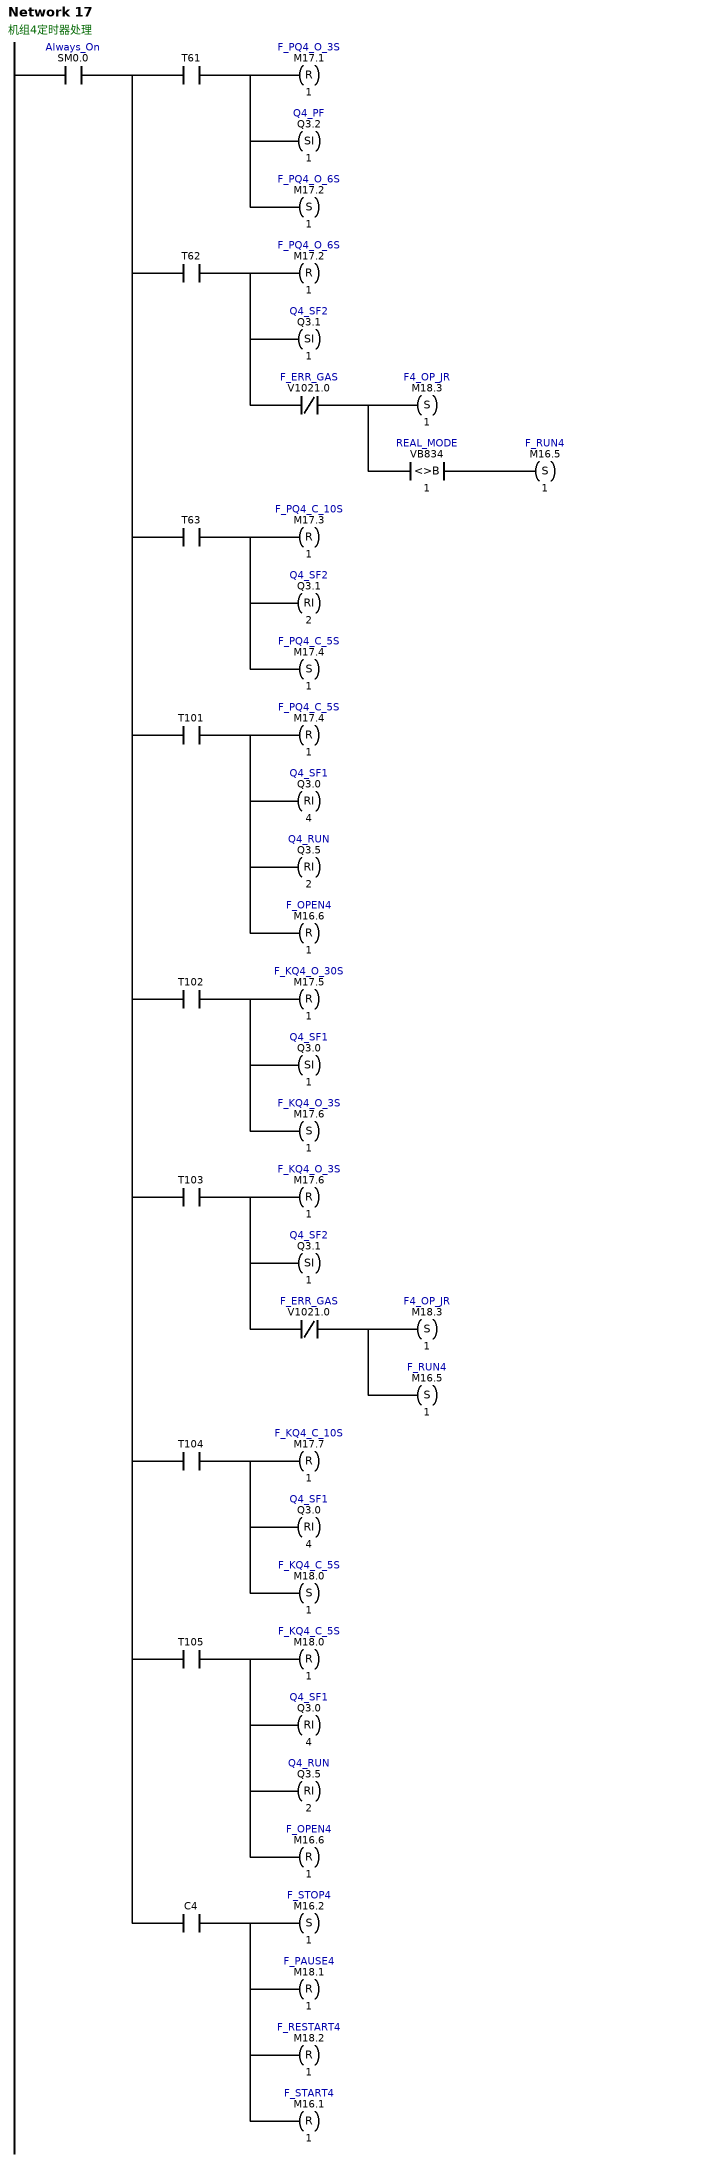
[picture p72: SBR7 networks 17-17]
Network 17
// 机组4定时器处理
LD     Always_On:SM0.0
LPS
A      T61
R      F_PQ4_O_3S:M17.1, 1
SI     Q4_PF:Q3.2, 1
S      F_PQ4_O_6S:M17.2, 1
LRD
A      T62
R      F_PQ4_O_6S:M17.2, 1
SI     Q4_SF2:Q3.1, 1
AN     F_ERR_GAS:V1021.0
S      F4_OP_JR:M18.3, 1
AB<>   REAL_MODE:VB834, 1
S      F_RUN4:M16.5, 1
LRD
LPS
A      T63
R      F_PQ4_C_10S:M17.3, 1
RI     Q4_SF2:Q3.1, 2
S      F_PQ4_C_5S:M17.4, 1
LRD
A      T101
R      F_PQ4_C_5S:M17.4, 1
RI     Q4_SF1:Q3.0, 4
RI     Q4_RUN:Q3.5, 2
R      F_OPEN4:M16.6, 1
LPP
A      T102
R      F_KQ4_O_30S:M17.5, 1
SI     Q4_SF1:Q3.0, 1
S      F_KQ4_O_3S:M17.6, 1
LRD
A      T103
R      F_KQ4_O_3S:M17.6, 1
SI     Q4_SF2:Q3.1, 1
AN     F_ERR_GAS:V1021.0
S      F4_OP_JR:M18.3, 1
S      F_RUN4:M16.5, 1
LPP
LPS
A      T104
R      F_KQ4_C_10S:M17.7, 1
RI     Q4_SF1:Q3.0, 4
S      F_KQ4_C_5S:M18.0, 1
LRD
A      T105
R      F_KQ4_C_5S:M18.0, 1
RI     Q4_SF1:Q3.0, 4
RI     Q4_RUN:Q3.5, 2
R      F_OPEN4:M16.6, 1
LPP
A      C4
S      F_STOP4:M16.2, 1
R      F_PAUSE4:M18.1, 1
R      F_RESTART4:M18.2, 1
R      F_START4:M16.1, 1
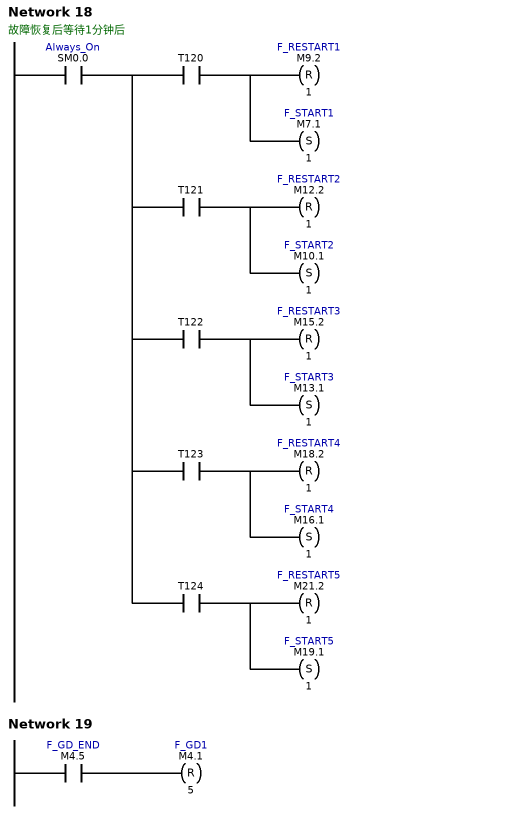
Network 18
// 故障恢复后等待1分钟后
LD     Always_On:SM0.0
LPS
A      T120
R      F_RESTART1:M9.2, 1
S      F_START1:M7.1, 1
LRD
A      T121
R      F_RESTART2:M12.2, 1
S      F_START2:M10.1, 1
LRD
A      T122
R      F_RESTART3:M15.2, 1
S      F_START3:M13.1, 1
LRD
A      T123
R      F_RESTART4:M18.2, 1
S      F_START4:M16.1, 1
LPP
A      T124
R      F_RESTART5:M21.2, 1
S      F_START5:M19.1, 1
Network 19
LD     F_GD_END:M4.5
R      F_GD1:M4.1, 5
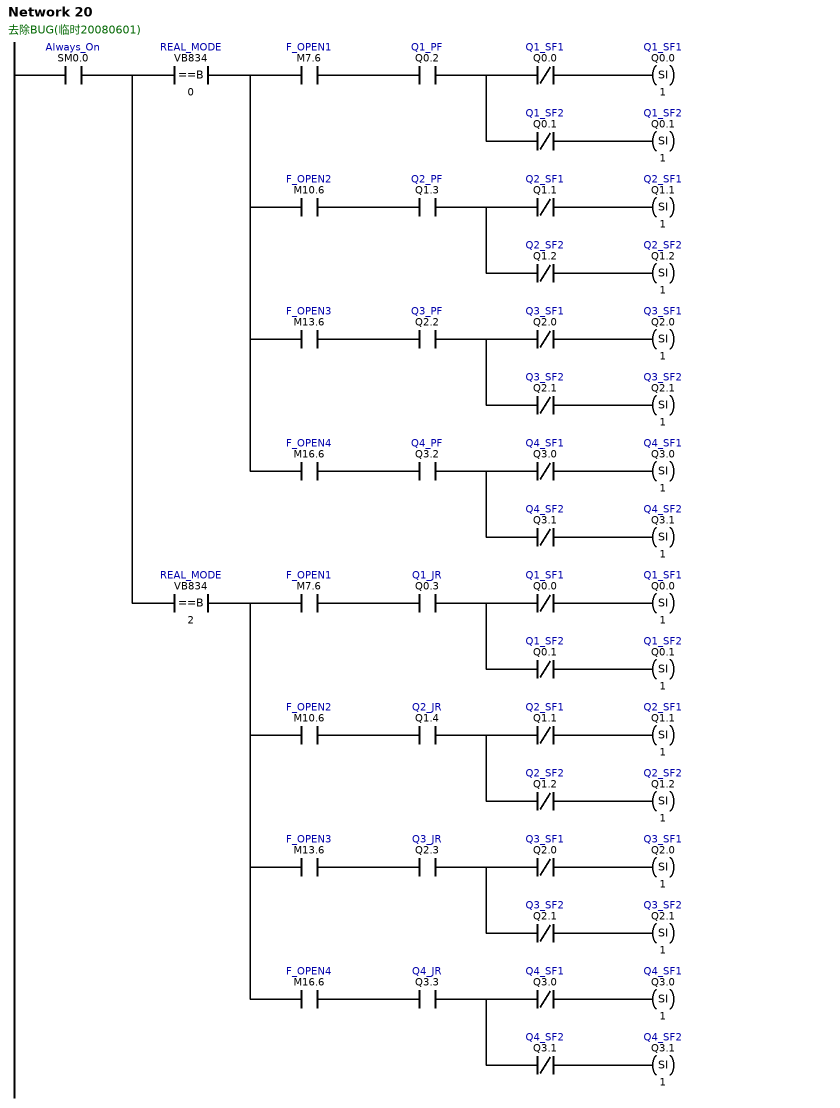
Network 20
// 去除BUG(临时20080601)
LD     Always_On:SM0.0
LPS
AB=    REAL_MODE:VB834, 0
LPS
A      F_OPEN1:M7.6
A      Q1_PF:Q0.2
LPS
AN     Q1_SF1:Q0.0
SI     Q1_SF1:Q0.0, 1
LPP
AN     Q1_SF2:Q0.1
SI     Q1_SF2:Q0.1, 1
LRD
A      F_OPEN2:M10.6
A      Q2_PF:Q1.3
LPS
AN     Q2_SF1:Q1.1
SI     Q2_SF1:Q1.1, 1
LPP
AN     Q2_SF2:Q1.2
SI     Q2_SF2:Q1.2, 1
LRD
A      F_OPEN3:M13.6
A      Q3_PF:Q2.2
LPS
AN     Q3_SF1:Q2.0
SI     Q3_SF1:Q2.0, 1
LPP
AN     Q3_SF2:Q2.1
SI     Q3_SF2:Q2.1, 1
LPP
A      F_OPEN4:M16.6
A      Q4_PF:Q3.2
LPS
AN     Q4_SF1:Q3.0
SI     Q4_SF1:Q3.0, 1
LPP
AN     Q4_SF2:Q3.1
SI     Q4_SF2:Q3.1, 1
LPP
AB=    REAL_MODE:VB834, 2
LPS
A      F_OPEN1:M7.6
A      Q1_JR:Q0.3
LPS
AN     Q1_SF1:Q0.0
SI     Q1_SF1:Q0.0, 1
LPP
AN     Q1_SF2:Q0.1
SI     Q1_SF2:Q0.1, 1
LRD
A      F_OPEN2:M10.6
A      Q2_JR:Q1.4
LPS
AN     Q2_SF1:Q1.1
SI     Q2_SF1:Q1.1, 1
LPP
AN     Q2_SF2:Q1.2
SI     Q2_SF2:Q1.2, 1
LRD
A      F_OPEN3:M13.6
A      Q3_JR:Q2.3
LPS
AN     Q3_SF1:Q2.0
SI     Q3_SF1:Q2.0, 1
LPP
AN     Q3_SF2:Q2.1
SI     Q3_SF2:Q2.1, 1
LPP
A      F_OPEN4:M16.6
A      Q4_JR:Q3.3
LPS
AN     Q4_SF1:Q3.0
SI     Q4_SF1:Q3.0, 1
LPP
AN     Q4_SF2:Q3.1
SI     Q4_SF2:Q3.1, 1
END_SUBROUTINE_BLOCK

SUBROUTINE_BLOCK 读EEPROM:SBR8
TITLE=
VAR
TEMP:DWORD;	// LD0 
END_VAR
BEGIN
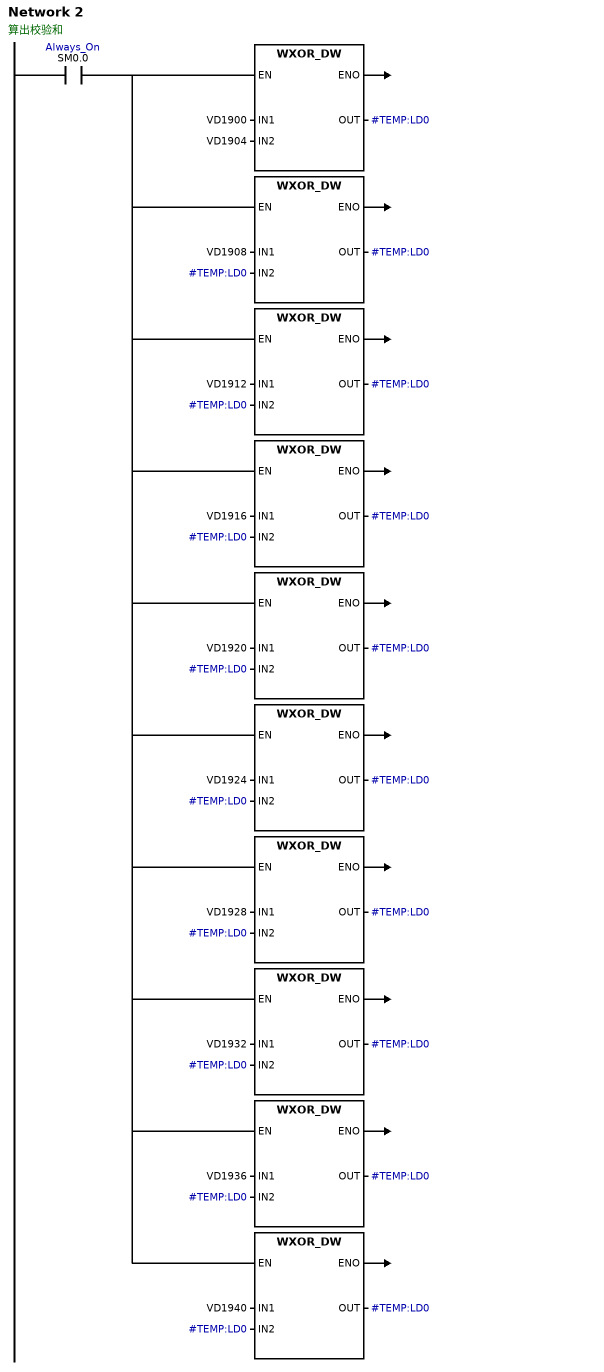
Network 2
// 算出校验和
LD     Always_On:SM0.0
MOVD   VD1900, #TEMP:LD0
XORD   VD1904, #TEMP:LD0
XORD   VD1908, #TEMP:LD0
XORD   VD1912, #TEMP:LD0
XORD   VD1916, #TEMP:LD0
XORD   VD1920, #TEMP:LD0
XORD   VD1924, #TEMP:LD0
XORD   VD1928, #TEMP:LD0
XORD   VD1932, #TEMP:LD0
XORD   VD1936, #TEMP:LD0
XORD   VD1940, #TEMP:LD0
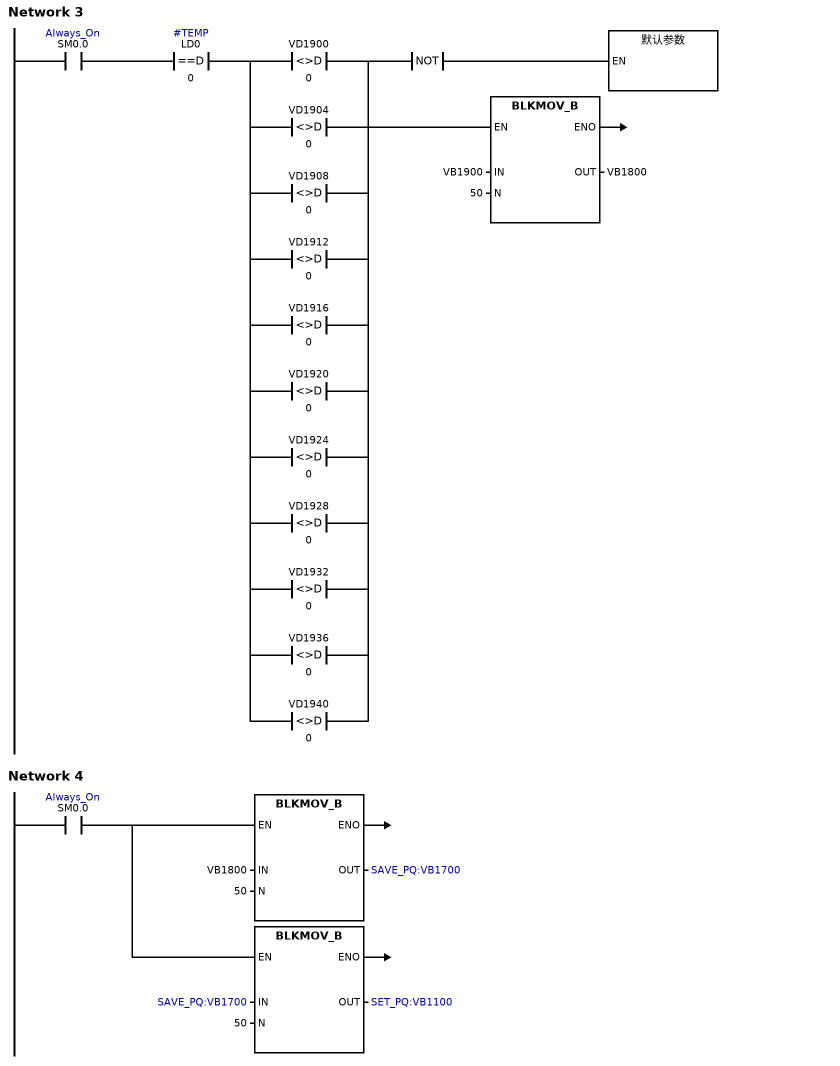
Network 3
LD     Always_On:SM0.0
AD=    #TEMP:LD0, 0
LDD<>  VD1900, 0
OD<>   VD1904, 0
OD<>   VD1908, 0
OD<>   VD1912, 0
OD<>   VD1916, 0
OD<>   VD1920, 0
OD<>   VD1924, 0
OD<>   VD1928, 0
OD<>   VD1932, 0
OD<>   VD1936, 0
OD<>   VD1940, 0
ALD
LPS
NOT
CALL   默认参数:SBR21
LPP
BMB    VB1900, VB1800, 50
Network 4
LD     Always_On:SM0.0
BMB    VB1800, SAVE_PQ:VB1700, 50
BMB    SAVE_PQ:VB1700, SET_PQ:VB1100, 50
END_SUBROUTINE_BLOCK

SUBROUTINE_BLOCK 定时器:SBR9
TITLE=
VAR
TEMP_W:WORD;	// LW0 
END_VAR
BEGIN
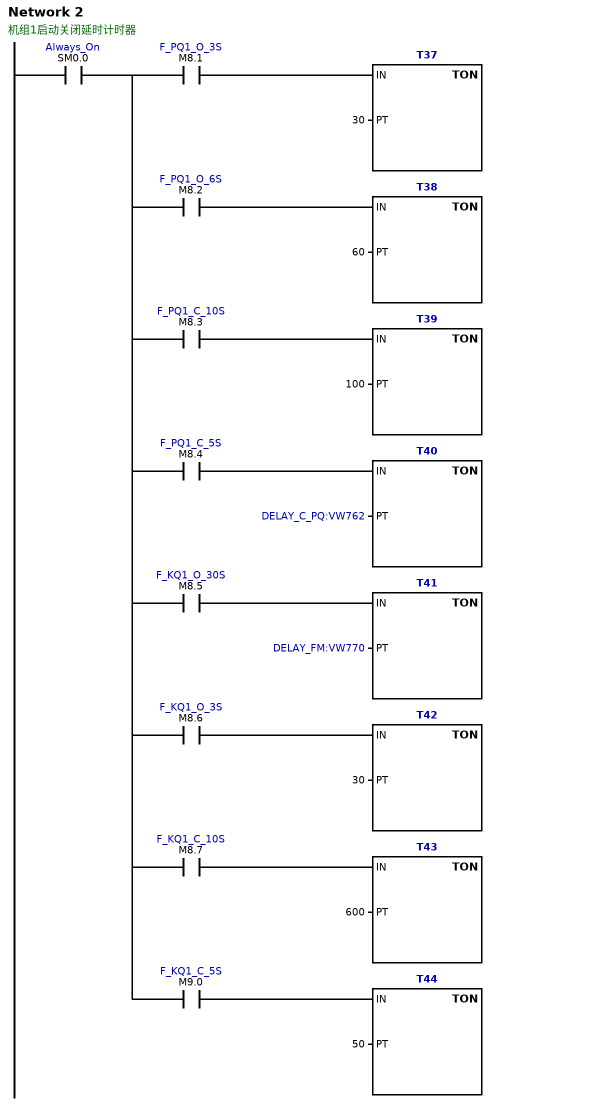
Network 2
// 机组1启动关闭延时计时器
LD     Always_On:SM0.0
LPS
A      F_PQ1_O_3S:M8.1
TON    T37, 30
LRD
A      F_PQ1_O_6S:M8.2
TON    T38, 60
LRD
A      F_PQ1_C_10S:M8.3
TON    T39, 100
LRD
A      F_PQ1_C_5S:M8.4
TON    T40, DELAY_C_PQ:VW762
LRD
A      F_KQ1_O_30S:M8.5
TON    T41, DELAY_FM:VW770
LRD
A      F_KQ1_O_3S:M8.6
TON    T42, 30
LRD
A      F_KQ1_C_10S:M8.7
TON    T43, 600
LPP
A      F_KQ1_C_5S:M9.0
TON    T44, 50
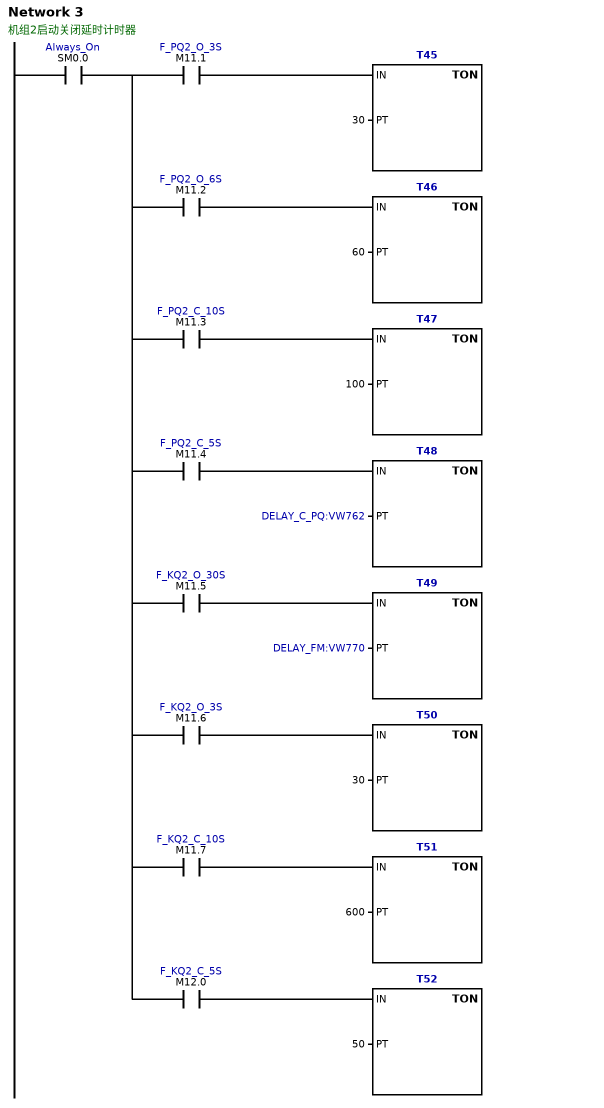
Network 3
// 机组2启动关闭延时计时器
LD     Always_On:SM0.0
LPS
A      F_PQ2_O_3S:M11.1
TON    T45, 30
LRD
A      F_PQ2_O_6S:M11.2
TON    T46, 60
LRD
A      F_PQ2_C_10S:M11.3
TON    T47, 100
LRD
A      F_PQ2_C_5S:M11.4
TON    T48, DELAY_C_PQ:VW762
LRD
A      F_KQ2_O_30S:M11.5
TON    T49, DELAY_FM:VW770
LRD
A      F_KQ2_O_3S:M11.6
TON    T50, 30
LRD
A      F_KQ2_C_10S:M11.7
TON    T51, 600
LPP
A      F_KQ2_C_5S:M12.0
TON    T52, 50
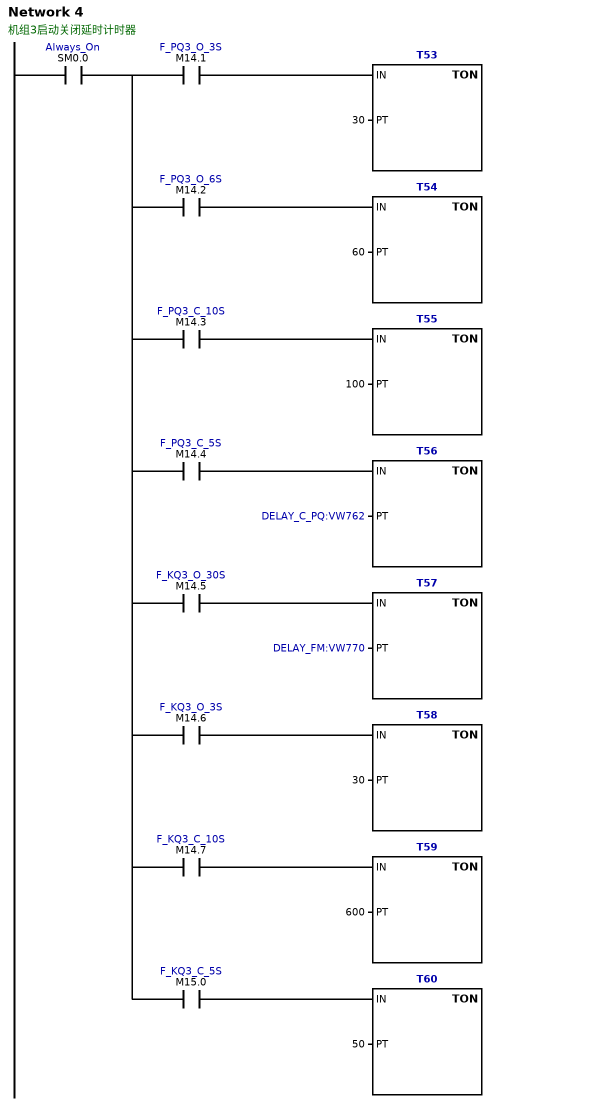
Network 4
// 机组3启动关闭延时计时器
LD     Always_On:SM0.0
LPS
A      F_PQ3_O_3S:M14.1
TON    T53, 30
LRD
A      F_PQ3_O_6S:M14.2
TON    T54, 60
LRD
A      F_PQ3_C_10S:M14.3
TON    T55, 100
LRD
A      F_PQ3_C_5S:M14.4
TON    T56, DELAY_C_PQ:VW762
LRD
A      F_KQ3_O_30S:M14.5
TON    T57, DELAY_FM:VW770
LRD
A      F_KQ3_O_3S:M14.6
TON    T58, 30
LRD
A      F_KQ3_C_10S:M14.7
TON    T59, 600
LPP
A      F_KQ3_C_5S:M15.0
TON    T60, 50
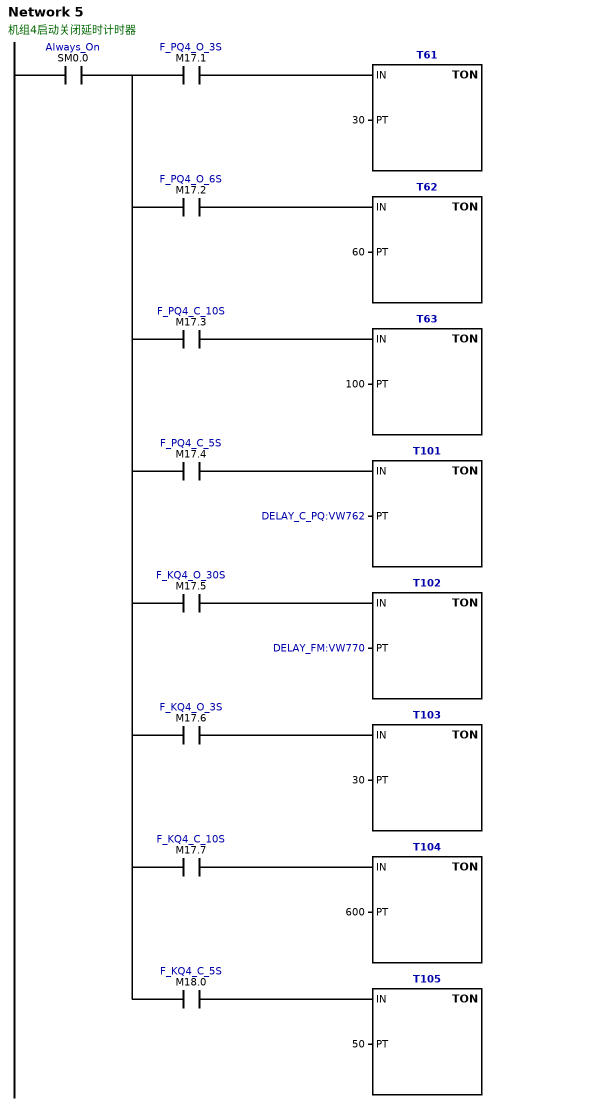
Network 5
// 机组4启动关闭延时计时器
LD     Always_On:SM0.0
LPS
A      F_PQ4_O_3S:M17.1
TON    T61, 30
LRD
A      F_PQ4_O_6S:M17.2
TON    T62, 60
LRD
A      F_PQ4_C_10S:M17.3
TON    T63, 100
LRD
A      F_PQ4_C_5S:M17.4
TON    T101, DELAY_C_PQ:VW762
LRD
A      F_KQ4_O_30S:M17.5
TON    T102, DELAY_FM:VW770
LRD
A      F_KQ4_O_3S:M17.6
TON    T103, 30
LRD
A      F_KQ4_C_10S:M17.7
TON    T104, 600
LPP
A      F_KQ4_C_5S:M18.0
TON    T105, 50
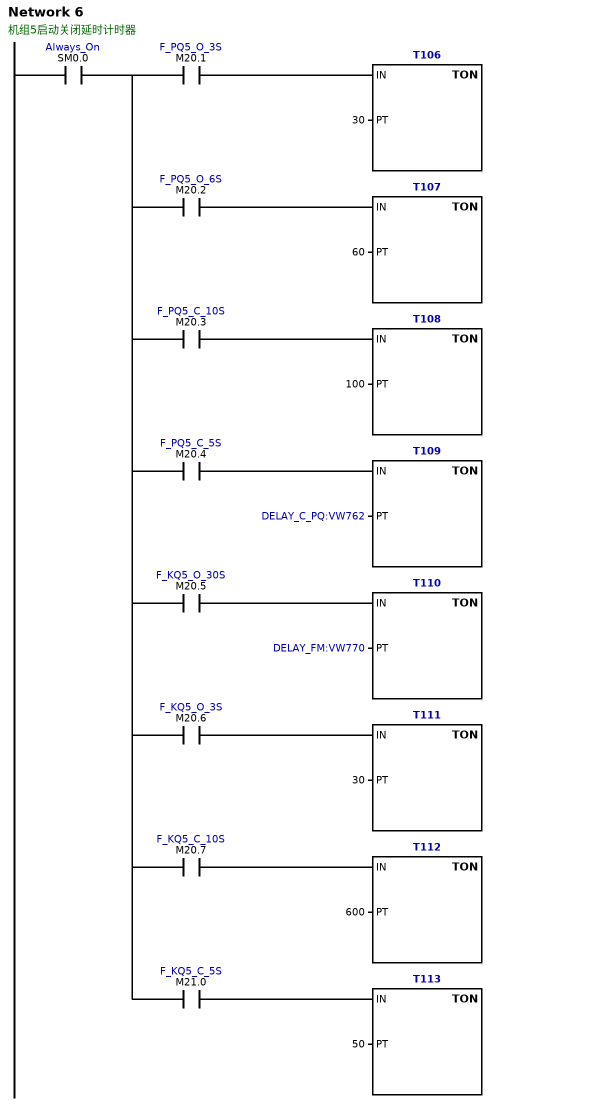
Network 6
// 机组5启动关闭延时计时器
LD     Always_On:SM0.0
LPS
A      F_PQ5_O_3S:M20.1
TON    T106, 30
LRD
A      F_PQ5_O_6S:M20.2
TON    T107, 60
LRD
A      F_PQ5_C_10S:M20.3
TON    T108, 100
LRD
A      F_PQ5_C_5S:M20.4
TON    T109, DELAY_C_PQ:VW762
LRD
A      F_KQ5_O_30S:M20.5
TON    T110, DELAY_FM:VW770
LRD
A      F_KQ5_O_3S:M20.6
TON    T111, 30
LRD
A      F_KQ5_C_10S:M20.7
TON    T112, 600
LPP
A      F_KQ5_C_5S:M21.0
TON    T113, 50
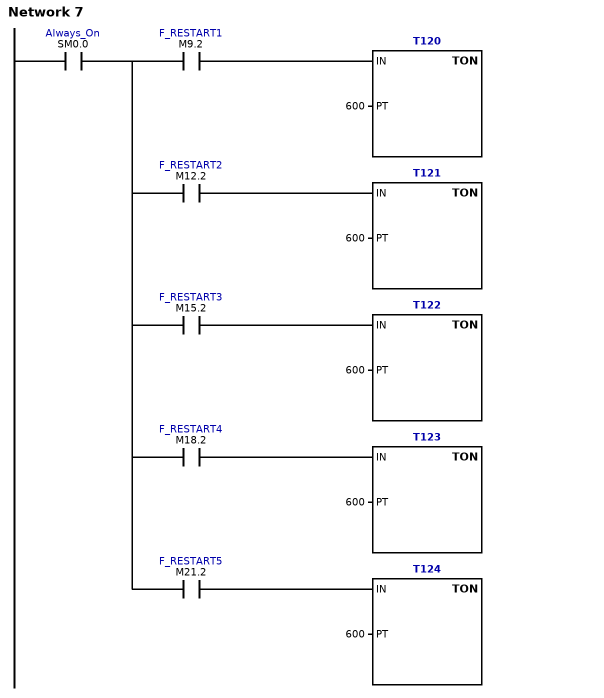
Network 7
LD     Always_On:SM0.0
LPS
A      F_RESTART1:M9.2
TON    T120, 600
LRD
A      F_RESTART2:M12.2
TON    T121, 600
LRD
A      F_RESTART3:M15.2
TON    T122, 600
LRD
A      F_RESTART4:M18.2
TON    T123, 600
LPP
A      F_RESTART5:M21.2
TON    T124, 600
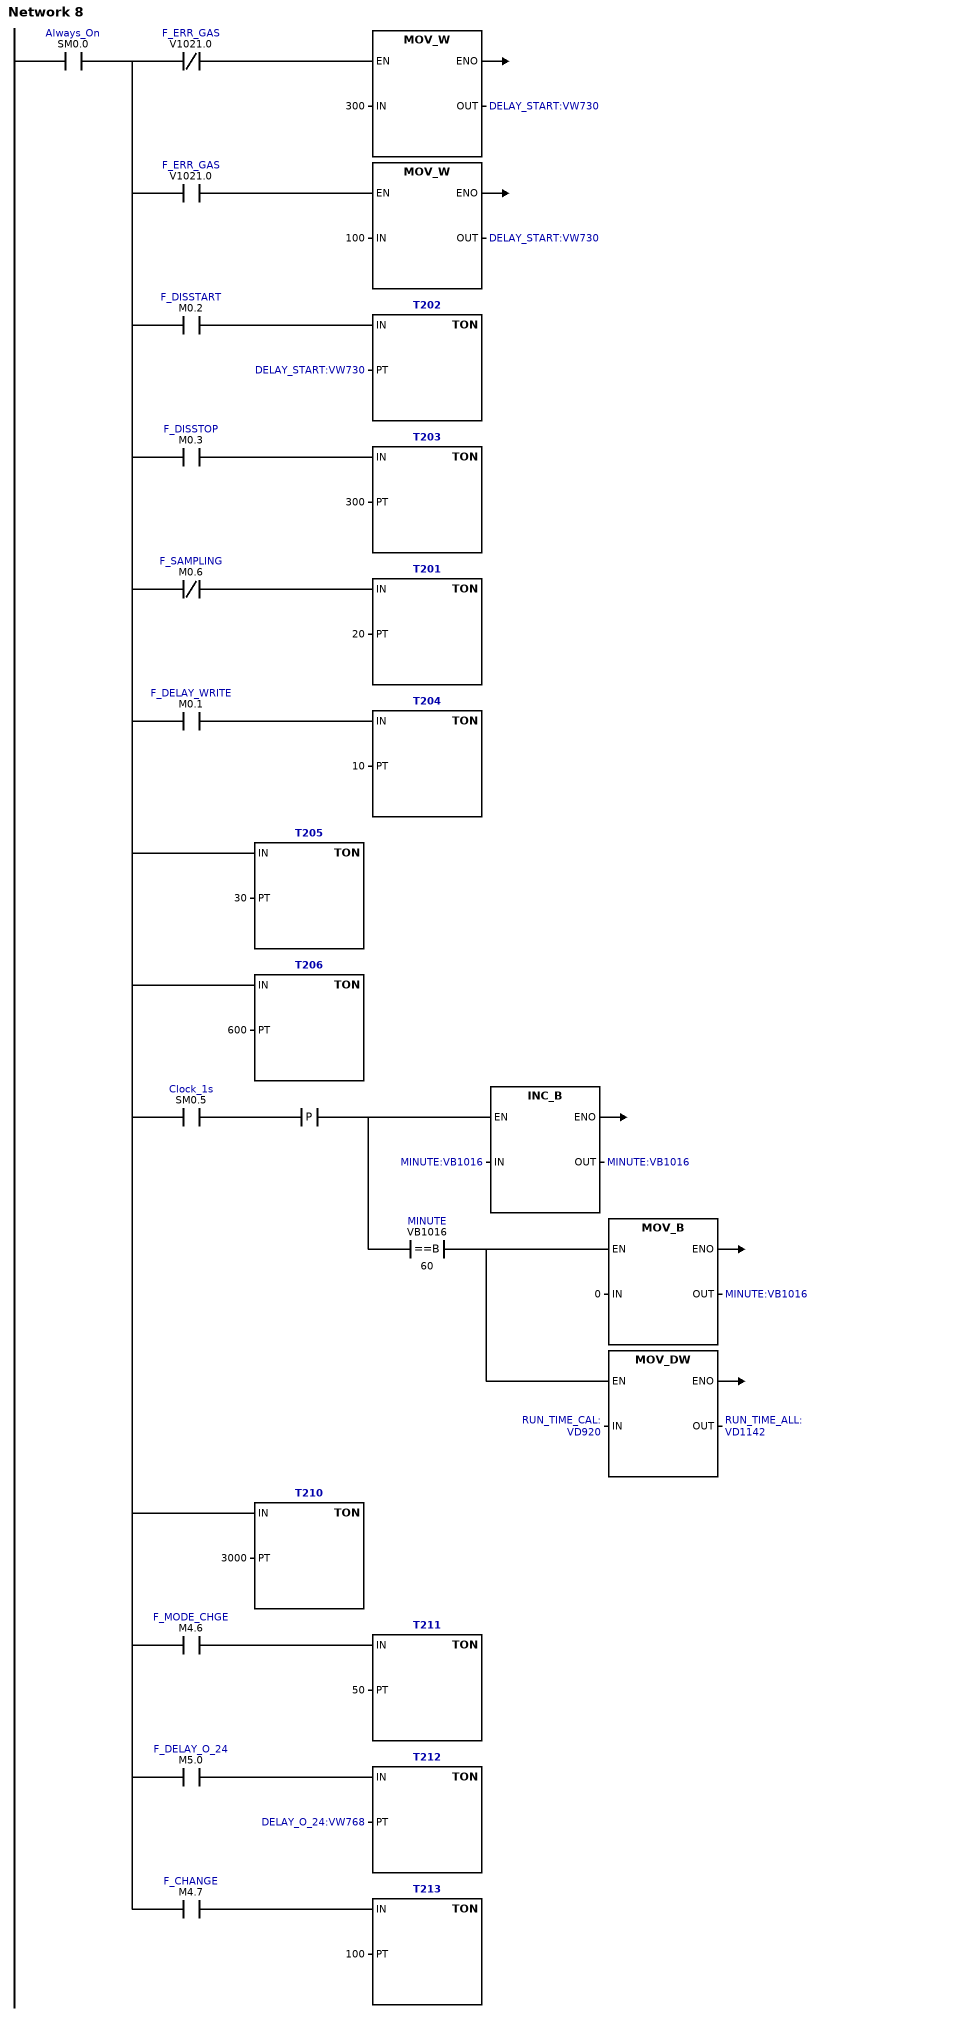
Network 8
LD     Always_On:SM0.0
LPS
AN     F_ERR_GAS:V1021.0
MOVW   300, DELAY_START:VW730
LRD
A      F_ERR_GAS:V1021.0
MOVW   100, DELAY_START:VW730
LRD
A      F_DISSTART:M0.2
TON    T202, DELAY_START:VW730
LRD
A      F_DISSTOP:M0.3
TON    T203, 300
LRD
AN     F_SAMPLING:M0.6
TON    T201, 20
LRD
A      F_DELAY_WRITE:M0.1
TON    T204, 10
LRD
TON    T205, 30
LRD
TON    T206, 600
LRD
A      Clock_1s:SM0.5
EU
INCB   MINUTE:VB1016
AB=    MINUTE:VB1016, 60
MOVB   0, MINUTE:VB1016
MOVD   RUN_TIME_CAL:VD920, RUN_TIME_ALL:VD1142
LPP
LPS
TON    T210, 3000
A      F_MODE_CHGE:M4.6
TON    T211, 50
LRD
A      F_DELAY_O_24:M5.0
TON    T212, DELAY_O_24:VW768
LPP
A      F_CHANGE:M4.7
TON    T213, 100
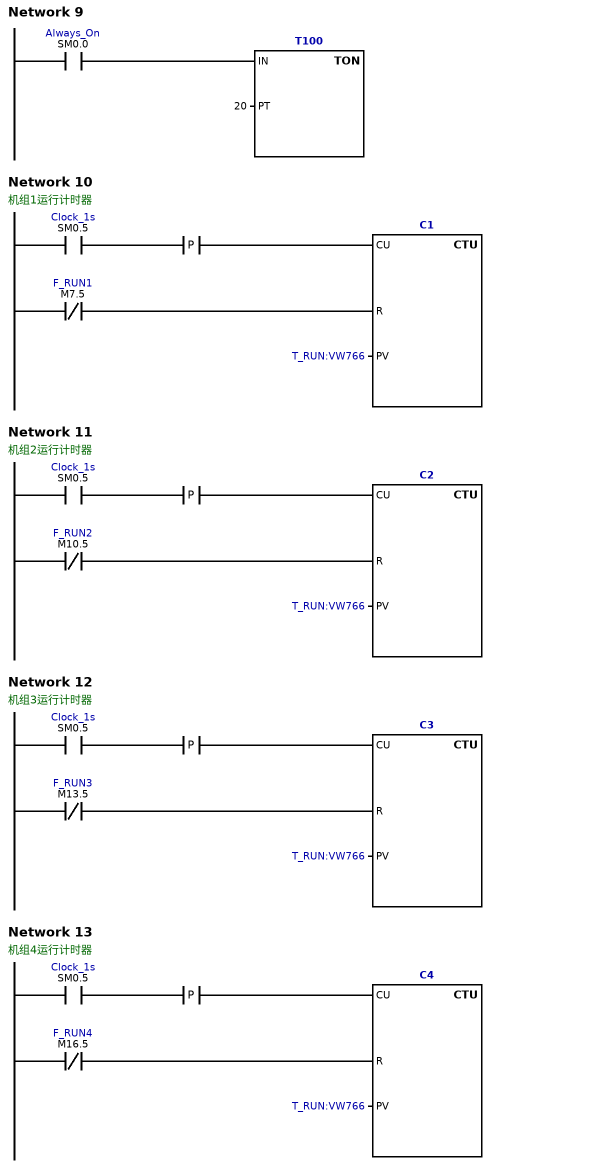
Network 9
LD     Always_On:SM0.0
TON    T100, 20
Network 10 //  
// 机组1运行计时器
LD     Clock_1s:SM0.5
EU
LDN    F_RUN1:M7.5
CTU    C1, T_RUN:VW766
Network 11 //  
// 机组2运行计时器
LD     Clock_1s:SM0.5
EU
LDN    F_RUN2:M10.5
CTU    C2, T_RUN:VW766
Network 12 //  
// 机组3运行计时器
LD     Clock_1s:SM0.5
EU
LDN    F_RUN3:M13.5
CTU    C3, T_RUN:VW766
Network 13 //  
// 机组4运行计时器
LD     Clock_1s:SM0.5
EU
LDN    F_RUN4:M16.5
CTU    C4, T_RUN:VW766
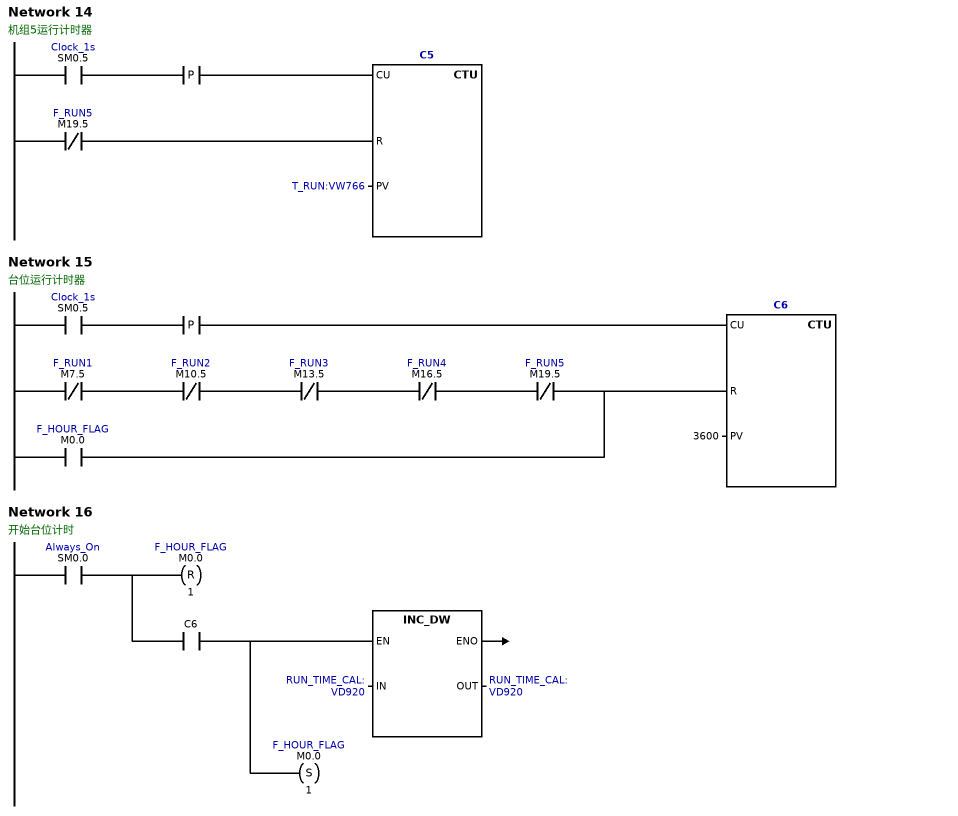
Network 14 //  
// 机组5运行计时器
LD     Clock_1s:SM0.5
EU
LDN    F_RUN5:M19.5
CTU    C5, T_RUN:VW766
Network 15 //  
// 台位运行计时器
LD     Clock_1s:SM0.5
EU
LDN    F_RUN1:M7.5
AN     F_RUN2:M10.5
AN     F_RUN3:M13.5
AN     F_RUN4:M16.5
AN     F_RUN5:M19.5
O      F_HOUR_FLAG:M0.0
CTU    C6, 3600
Network 16
// 开始台位计时
LD     Always_On:SM0.0
R      F_HOUR_FLAG:M0.0, 1
A      C6
INCD   RUN_TIME_CAL:VD920
S      F_HOUR_FLAG:M0.0, 1
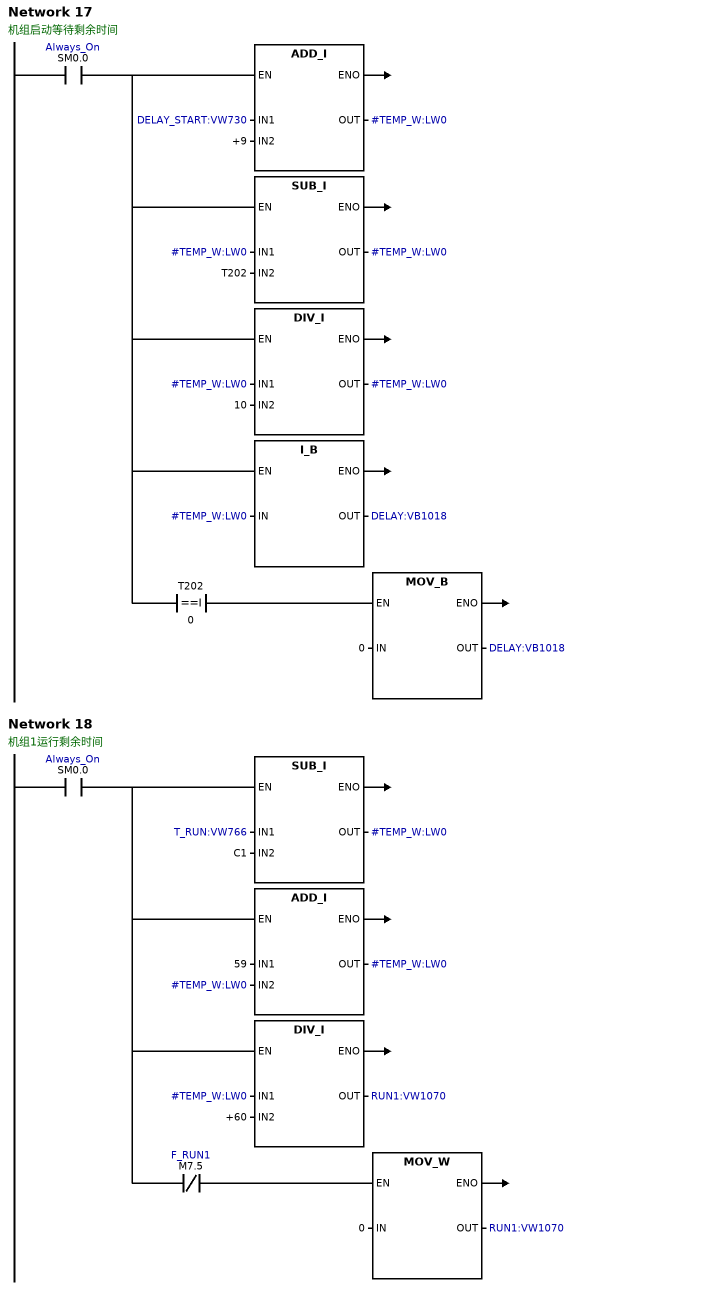
Network 17
// 机组启动等待剩余时间
LD     Always_On:SM0.0
MOVW   DELAY_START:VW730, #TEMP_W:LW0
+I     +9, #TEMP_W:LW0
-I     T202, #TEMP_W:LW0
/I     10, #TEMP_W:LW0
ITB    #TEMP_W:LW0, DELAY:VB1018
AW=    T202, 0
MOVB   0, DELAY:VB1018
Network 18
// 机组1运行剩余时间
LD     Always_On:SM0.0
MOVW   T_RUN:VW766, #TEMP_W:LW0
-I     C1, #TEMP_W:LW0
+I     59, #TEMP_W:LW0
MOVW   #TEMP_W:LW0, RUN1:VW1070
/I     +60, RUN1:VW1070
AN     F_RUN1:M7.5
MOVW   0, RUN1:VW1070
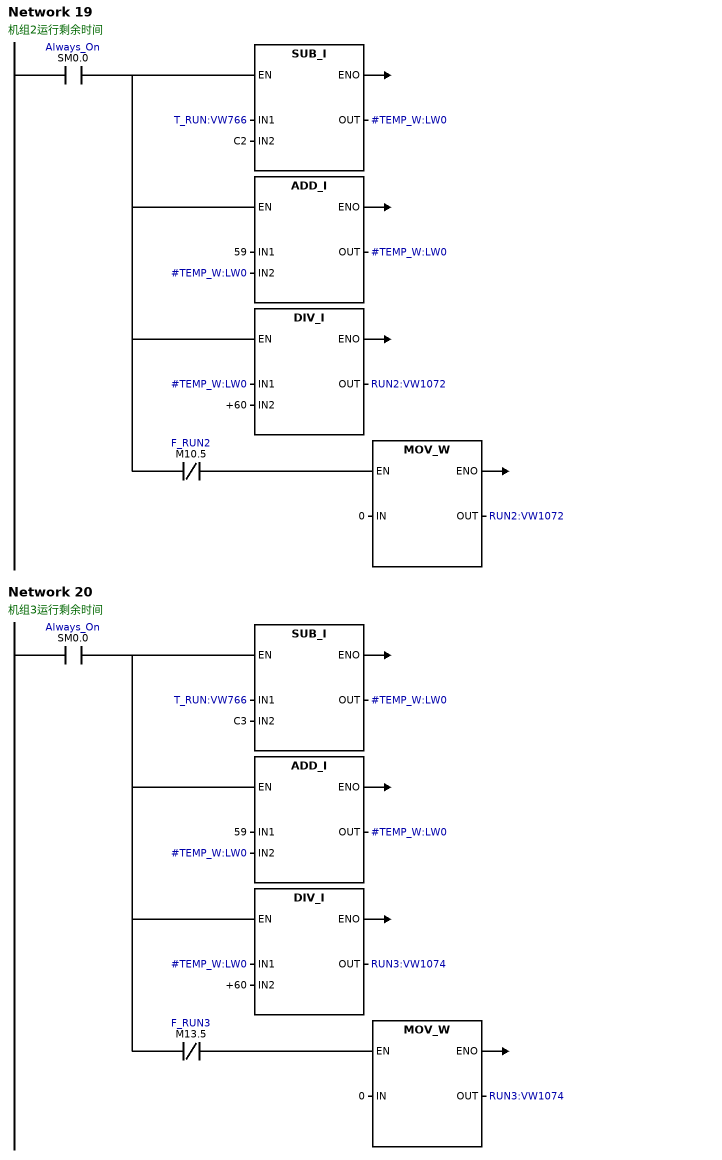
Network 19
// 机组2运行剩余时间
LD     Always_On:SM0.0
MOVW   T_RUN:VW766, #TEMP_W:LW0
-I     C2, #TEMP_W:LW0
+I     59, #TEMP_W:LW0
MOVW   #TEMP_W:LW0, RUN2:VW1072
/I     +60, RUN2:VW1072
AN     F_RUN2:M10.5
MOVW   0, RUN2:VW1072
Network 20
// 机组3运行剩余时间
LD     Always_On:SM0.0
MOVW   T_RUN:VW766, #TEMP_W:LW0
-I     C3, #TEMP_W:LW0
+I     59, #TEMP_W:LW0
MOVW   #TEMP_W:LW0, RUN3:VW1074
/I     +60, RUN3:VW1074
AN     F_RUN3:M13.5
MOVW   0, RUN3:VW1074
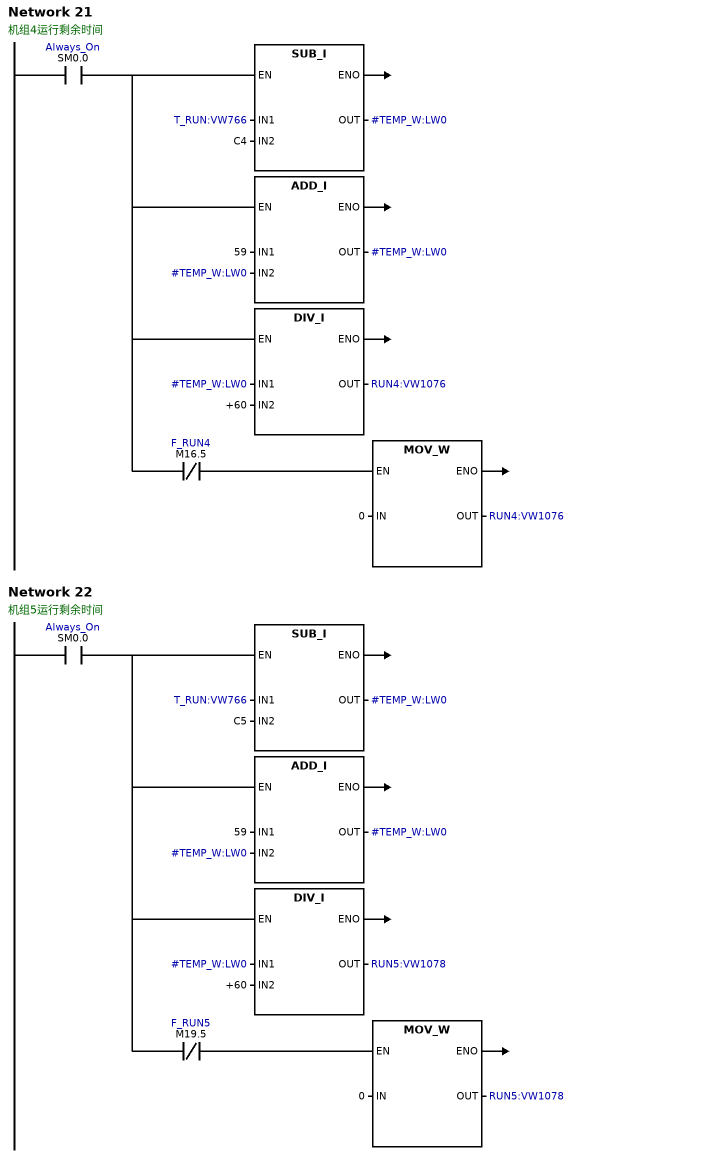
Network 21
// 机组4运行剩余时间
LD     Always_On:SM0.0
MOVW   T_RUN:VW766, #TEMP_W:LW0
-I     C4, #TEMP_W:LW0
+I     59, #TEMP_W:LW0
MOVW   #TEMP_W:LW0, RUN4:VW1076
/I     +60, RUN4:VW1076
AN     F_RUN4:M16.5
MOVW   0, RUN4:VW1076
Network 22
// 机组5运行剩余时间
LD     Always_On:SM0.0
MOVW   T_RUN:VW766, #TEMP_W:LW0
-I     C5, #TEMP_W:LW0
+I     59, #TEMP_W:LW0
MOVW   #TEMP_W:LW0, RUN5:VW1078
/I     +60, RUN5:VW1078
AN     F_RUN5:M19.5
MOVW   0, RUN5:VW1078
END_SUBROUTINE_BLOCK

SUBROUTINE_BLOCK 温度处理:SBR10
TITLE=
VAR
TEMP_T:WORD;	// LW0 
END_VAR
BEGIN
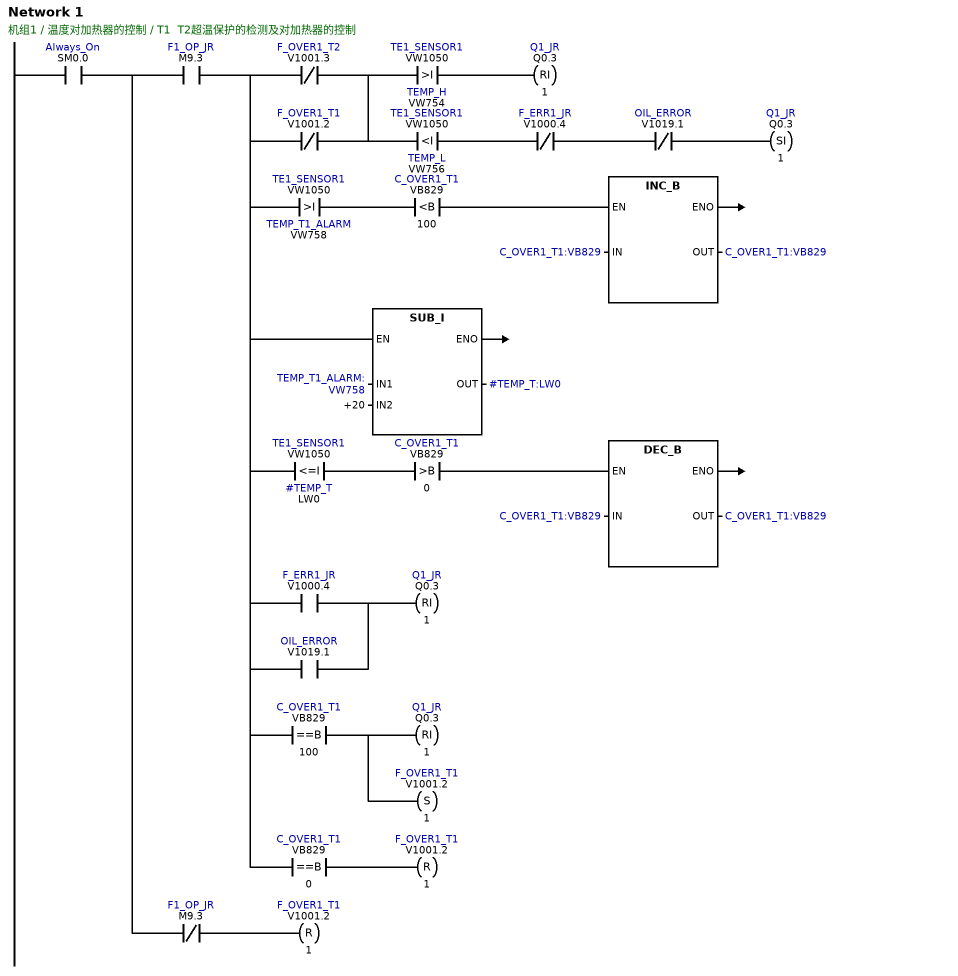
Network 1
// 机组1
// 温度对加热器的控制
// T1  T2超温保护的检测及对加热器的控制
LD     Always_On:SM0.0
LPS
A      F1_OP_JR:M9.3
LPS
LDN    F_OVER1_T2:V1001.3
ON     F_OVER1_T1:V1001.2
ALD
LPS
AW>    TE1_SENSOR1:VW1050, TEMP_H:VW754
RI     Q1_JR:Q0.3, 1
LPP
AW<    TE1_SENSOR1:VW1050, TEMP_L:VW756
AN     F_ERR1_JR:V1000.4
AN     OIL_ERROR:V1019.1
SI     Q1_JR:Q0.3, 1
LRD
LPS
AW>    TE1_SENSOR1:VW1050, TEMP_T1_ALARM:VW758
AB<    C_OVER1_T1:VB829, 100
INCB   C_OVER1_T1:VB829
LRD
MOVW   TEMP_T1_ALARM:VW758, #TEMP_T:LW0
-I     +20, #TEMP_T:LW0
LPP
AW<=   TE1_SENSOR1:VW1050, #TEMP_T:LW0
AB>    C_OVER1_T1:VB829, 0
DECB   C_OVER1_T1:VB829
LRD
LD     F_ERR1_JR:V1000.4
O      OIL_ERROR:V1019.1
ALD
RI     Q1_JR:Q0.3, 1
LRD
AB=    C_OVER1_T1:VB829, 100
RI     Q1_JR:Q0.3, 1
S      F_OVER1_T1:V1001.2, 1
LPP
AB=    C_OVER1_T1:VB829, 0
R      F_OVER1_T1:V1001.2, 1
LPP
AN     F1_OP_JR:M9.3
R      F_OVER1_T1:V1001.2, 1
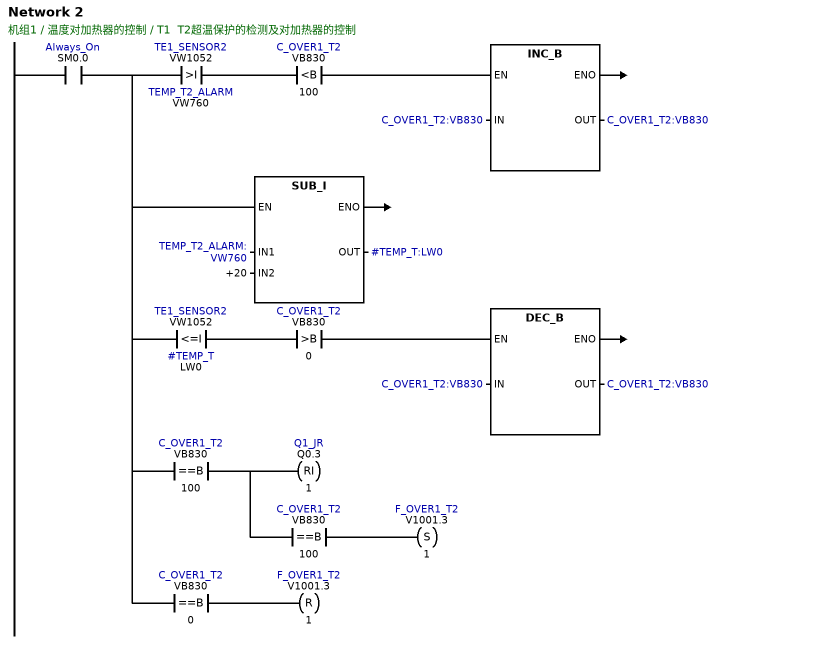
Network 2
// 机组1
// 温度对加热器的控制
// T1  T2超温保护的检测及对加热器的控制
LD     Always_On:SM0.0
LPS
AW>    TE1_SENSOR2:VW1052, TEMP_T2_ALARM:VW760
AB<    C_OVER1_T2:VB830, 100
INCB   C_OVER1_T2:VB830
LRD
MOVW   TEMP_T2_ALARM:VW760, #TEMP_T:LW0
-I     +20, #TEMP_T:LW0
LRD
AW<=   TE1_SENSOR2:VW1052, #TEMP_T:LW0
AB>    C_OVER1_T2:VB830, 0
DECB   C_OVER1_T2:VB830
LRD
AB=    C_OVER1_T2:VB830, 100
RI     Q1_JR:Q0.3, 1
AB=    C_OVER1_T2:VB830, 100
S      F_OVER1_T2:V1001.3, 1
LPP
AB=    C_OVER1_T2:VB830, 0
R      F_OVER1_T2:V1001.3, 1
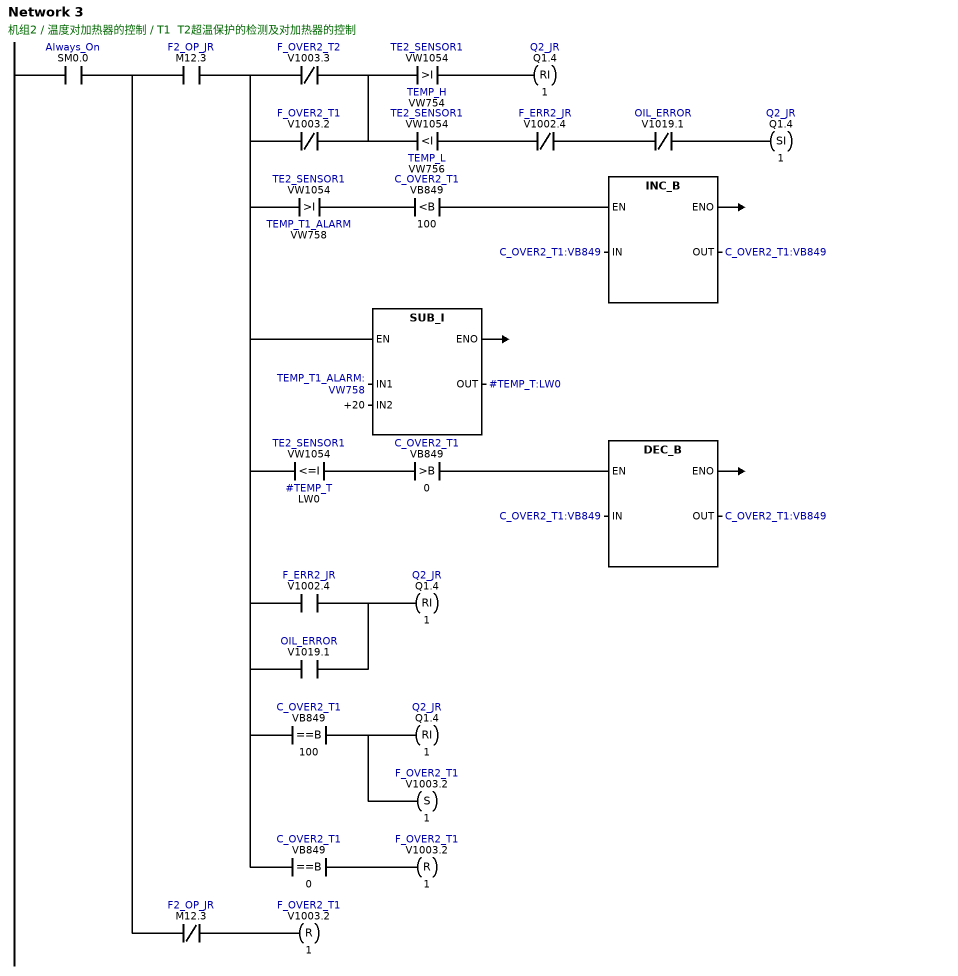
Network 3
// 机组2
// 温度对加热器的控制
// T1  T2超温保护的检测及对加热器的控制
LD     Always_On:SM0.0
LPS
A      F2_OP_JR:M12.3
LPS
LDN    F_OVER2_T2:V1003.3
ON     F_OVER2_T1:V1003.2
ALD
LPS
AW>    TE2_SENSOR1:VW1054, TEMP_H:VW754
RI     Q2_JR:Q1.4, 1
LPP
AW<    TE2_SENSOR1:VW1054, TEMP_L:VW756
AN     F_ERR2_JR:V1002.4
AN     OIL_ERROR:V1019.1
SI     Q2_JR:Q1.4, 1
LRD
LPS
AW>    TE2_SENSOR1:VW1054, TEMP_T1_ALARM:VW758
AB<    C_OVER2_T1:VB849, 100
INCB   C_OVER2_T1:VB849
LRD
MOVW   TEMP_T1_ALARM:VW758, #TEMP_T:LW0
-I     +20, #TEMP_T:LW0
LPP
AW<=   TE2_SENSOR1:VW1054, #TEMP_T:LW0
AB>    C_OVER2_T1:VB849, 0
DECB   C_OVER2_T1:VB849
LRD
LD     F_ERR2_JR:V1002.4
O      OIL_ERROR:V1019.1
ALD
RI     Q2_JR:Q1.4, 1
LRD
AB=    C_OVER2_T1:VB849, 100
RI     Q2_JR:Q1.4, 1
S      F_OVER2_T1:V1003.2, 1
LPP
AB=    C_OVER2_T1:VB849, 0
R      F_OVER2_T1:V1003.2, 1
LPP
AN     F2_OP_JR:M12.3
R      F_OVER2_T1:V1003.2, 1
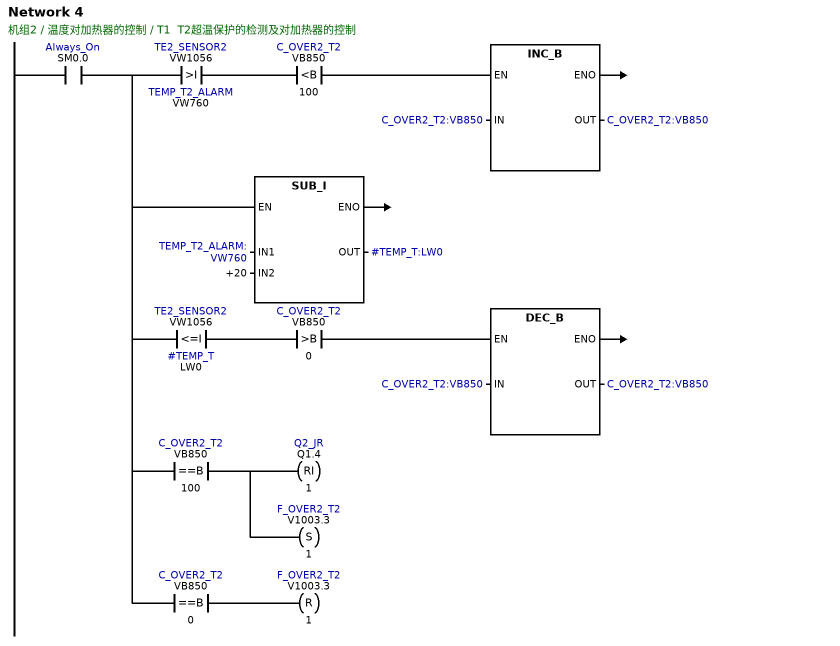
Network 4
// 机组2
// 温度对加热器的控制
// T1  T2超温保护的检测及对加热器的控制
LD     Always_On:SM0.0
LPS
AW>    TE2_SENSOR2:VW1056, TEMP_T2_ALARM:VW760
AB<    C_OVER2_T2:VB850, 100
INCB   C_OVER2_T2:VB850
LRD
MOVW   TEMP_T2_ALARM:VW760, #TEMP_T:LW0
-I     +20, #TEMP_T:LW0
LRD
AW<=   TE2_SENSOR2:VW1056, #TEMP_T:LW0
AB>    C_OVER2_T2:VB850, 0
DECB   C_OVER2_T2:VB850
LRD
AB=    C_OVER2_T2:VB850, 100
RI     Q2_JR:Q1.4, 1
S      F_OVER2_T2:V1003.3, 1
LPP
AB=    C_OVER2_T2:VB850, 0
R      F_OVER2_T2:V1003.3, 1
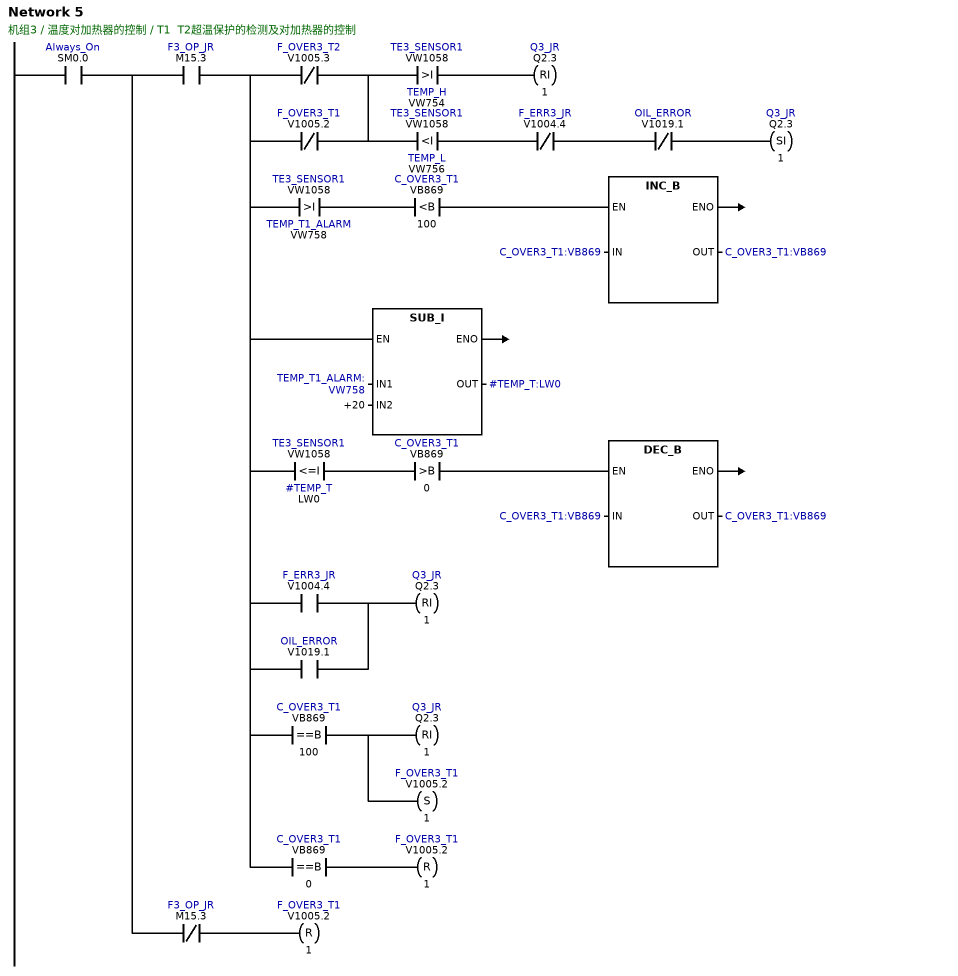
Network 5
// 机组3
// 温度对加热器的控制
// T1  T2超温保护的检测及对加热器的控制
LD     Always_On:SM0.0
LPS
A      F3_OP_JR:M15.3
LPS
LDN    F_OVER3_T2:V1005.3
ON     F_OVER3_T1:V1005.2
ALD
LPS
AW>    TE3_SENSOR1:VW1058, TEMP_H:VW754
RI     Q3_JR:Q2.3, 1
LPP
AW<    TE3_SENSOR1:VW1058, TEMP_L:VW756
AN     F_ERR3_JR:V1004.4
AN     OIL_ERROR:V1019.1
SI     Q3_JR:Q2.3, 1
LRD
LPS
AW>    TE3_SENSOR1:VW1058, TEMP_T1_ALARM:VW758
AB<    C_OVER3_T1:VB869, 100
INCB   C_OVER3_T1:VB869
LRD
MOVW   TEMP_T1_ALARM:VW758, #TEMP_T:LW0
-I     +20, #TEMP_T:LW0
LPP
AW<=   TE3_SENSOR1:VW1058, #TEMP_T:LW0
AB>    C_OVER3_T1:VB869, 0
DECB   C_OVER3_T1:VB869
LRD
LD     F_ERR3_JR:V1004.4
O      OIL_ERROR:V1019.1
ALD
RI     Q3_JR:Q2.3, 1
LRD
AB=    C_OVER3_T1:VB869, 100
RI     Q3_JR:Q2.3, 1
S      F_OVER3_T1:V1005.2, 1
LPP
AB=    C_OVER3_T1:VB869, 0
R      F_OVER3_T1:V1005.2, 1
LPP
AN     F3_OP_JR:M15.3
R      F_OVER3_T1:V1005.2, 1
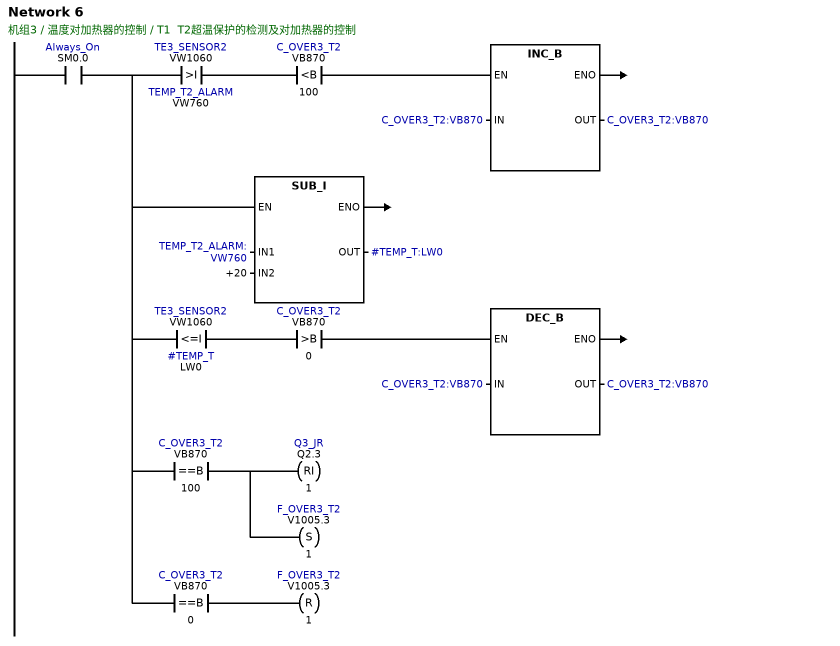
Network 6
// 机组3
// 温度对加热器的控制
// T1  T2超温保护的检测及对加热器的控制
LD     Always_On:SM0.0
LPS
AW>    TE3_SENSOR2:VW1060, TEMP_T2_ALARM:VW760
AB<    C_OVER3_T2:VB870, 100
INCB   C_OVER3_T2:VB870
LRD
MOVW   TEMP_T2_ALARM:VW760, #TEMP_T:LW0
-I     +20, #TEMP_T:LW0
LRD
AW<=   TE3_SENSOR2:VW1060, #TEMP_T:LW0
AB>    C_OVER3_T2:VB870, 0
DECB   C_OVER3_T2:VB870
LRD
AB=    C_OVER3_T2:VB870, 100
RI     Q3_JR:Q2.3, 1
S      F_OVER3_T2:V1005.3, 1
LPP
AB=    C_OVER3_T2:VB870, 0
R      F_OVER3_T2:V1005.3, 1
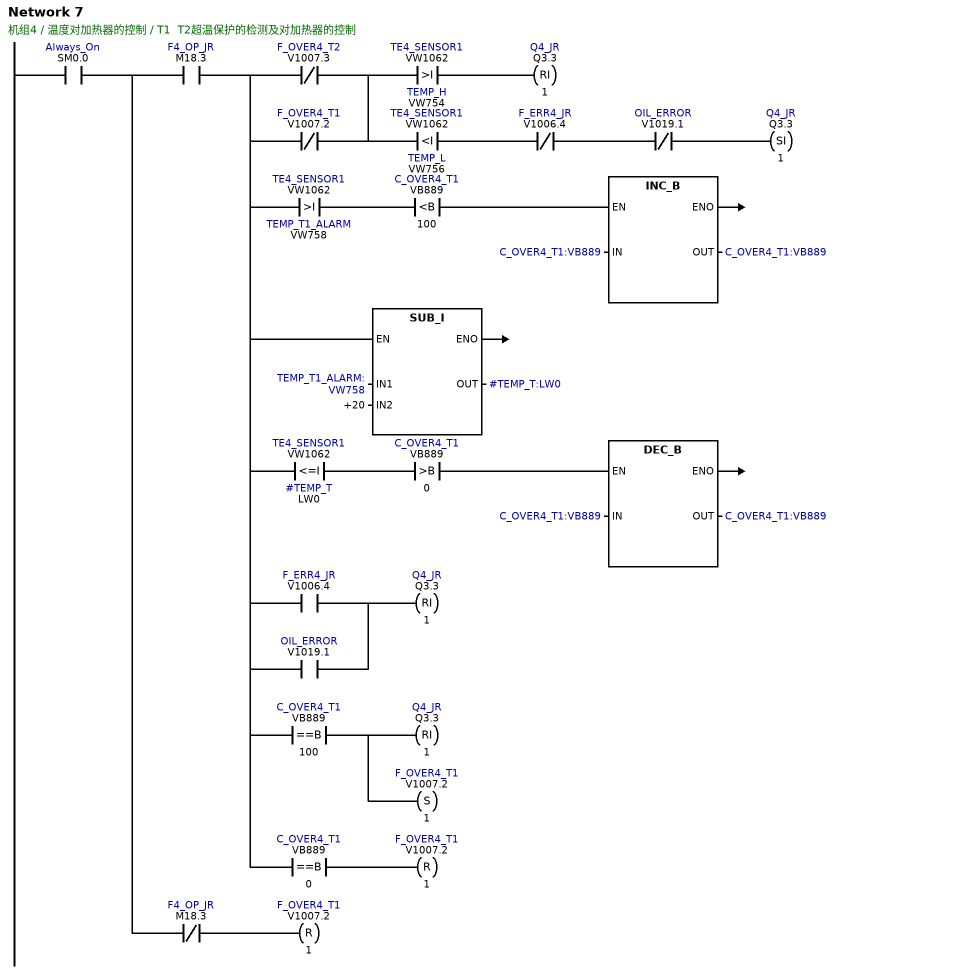
Network 7
// 机组4
// 温度对加热器的控制
// T1  T2超温保护的检测及对加热器的控制
LD     Always_On:SM0.0
LPS
A      F4_OP_JR:M18.3
LPS
LDN    F_OVER4_T2:V1007.3
ON     F_OVER4_T1:V1007.2
ALD
LPS
AW>    TE4_SENSOR1:VW1062, TEMP_H:VW754
RI     Q4_JR:Q3.3, 1
LPP
AW<    TE4_SENSOR1:VW1062, TEMP_L:VW756
AN     F_ERR4_JR:V1006.4
AN     OIL_ERROR:V1019.1
SI     Q4_JR:Q3.3, 1
LRD
LPS
AW>    TE4_SENSOR1:VW1062, TEMP_T1_ALARM:VW758
AB<    C_OVER4_T1:VB889, 100
INCB   C_OVER4_T1:VB889
LRD
MOVW   TEMP_T1_ALARM:VW758, #TEMP_T:LW0
-I     +20, #TEMP_T:LW0
LPP
AW<=   TE4_SENSOR1:VW1062, #TEMP_T:LW0
AB>    C_OVER4_T1:VB889, 0
DECB   C_OVER4_T1:VB889
LRD
LD     F_ERR4_JR:V1006.4
O      OIL_ERROR:V1019.1
ALD
RI     Q4_JR:Q3.3, 1
LRD
AB=    C_OVER4_T1:VB889, 100
RI     Q4_JR:Q3.3, 1
S      F_OVER4_T1:V1007.2, 1
LPP
AB=    C_OVER4_T1:VB889, 0
R      F_OVER4_T1:V1007.2, 1
LPP
AN     F4_OP_JR:M18.3
R      F_OVER4_T1:V1007.2, 1
